ABB RobotStudio station: ExternalGuidedMotion.rsstn

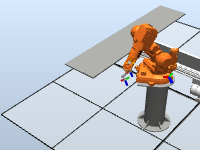
Station E459_norbert (saved by RobotStudio format 3)
Controller IRB140_6kg_0.81m_typeC_1, task T_ROB1: task frame (RAPID world) sits at (10, 680, 720) mm, rotated rx 0 ry 0 rz -30 deg in the station
Controller NorbertEGMVirtuel, task T_ROB1: task frame (RAPID world) sits at (-305, -752, 720) mm, rotated rx 0 ry 0 rz 30 deg in the station
Controller NorbertEGMVirtuel
  mechanical unit ROB_1: Norbert, 6 joints, base frame (0, 0, 0) mm
  mechanical unit CNV1: ?, 1 joints, base frame (0, 0, 0) mm
Controller IRB140_6kg_0.81m_typeC_1
  mechanical unit ROB_1: Rudolf, 6 joints, base frame (0, 0, 0) mm
Layout (positions relative to the parent item):
  - PedestalR [part, from Libraries\Pedestal.rslib] at (10, 680, 0) mm, rotated rx 0 ry 0 rz 150 deg
  - PedestalN [part, from Libraries\Pedestal.rslib] at (-305, -752, 0) mm, rotated rx 0 ry 0 rz -150 deg
  - Windowtable [part]
  - BordR [part, from Libraries\Desk.rslib] at (193.4, 1497.66, 0) mm, rotated rx 0 ry 0 rz -120 deg
  - Norbert [mechanism, from Libraries\IRB140_6_81_C_01.rslib] at (-305, -752, 720) mm, rotated rx 0 ry 0 rz 30 deg; joint values [-2.4777, 0.5946, 0.434, -2.4087, -0.8902, -0.8561] (rad or m)
  - Rudolf [mechanism, from Libraries\IRB140_6_81_C_01.rslib] at (10, 680, 720) mm, rotated rx 0 ry 0 rz -30 deg; joint values [1.249, 0.6446, -0.2193, 0, 1.1455, 1.249] (rad or m)
  - Conveyor [part, from Libraries\Conveyor.rslib] at (-998.97, -64.27, 615.81) mm, rotated rx 90 ry 0 rz -90 deg
  - tSuctionCup [mechanism, from Libraries\tSuctionCup.rslib] at (-444.43, -1188.19, 990.31) mm, rotated rx -146.84 ry 1 rz -95.37 deg
  - Conveyor_2 [part, from Libraries\Conveyor_1.rslib] at (-998.97, -64.27, 615.81) mm, rotated rx 90 ry 0 rz -90 deg
Attachment: BordR is attached to PedestalR
Attachment: tSuctionCup is attached to Norbert / Link6
Station signals: DI doClose, DI doOpen
Station logic (signal -> signal, property => property):
  NorbertEGMVirtuel.doOpen -> ?.diOpen
  NorbertEGMVirtuel.doClose -> ?.diClose
  ?.doClosed -> NorbertEGMVirtuel.diClosed
Targets, tools, work objects and paths stored in the station, written as RAPID:
! task T_ROB1
MODULE EGM_test_analog
  VAR signalao ao_MoveX;
  VAR signalao ao_MoveY;
  VAR signalao ao_MoveZ;
  TASK PERS loaddata load1:=[5,[0,1,0],[1,0,0,0],0,0,0];
  VAR signalao ao_RotX;
  VAR signalao ao_RotY;
  VAR signalao ao_RotZ;
ENDMODULE

! task T_ROB1
MODULE ExternalGuidedMotion
  TASK PERS tooldata tSuctionCup:=[TRUE,[[120,0,57],[0.707106624,-0.000000155,-0.000000251,0.707106939]],[1,[0,0,1],[1,0,0,0],0,0,0]];
  TASK PERS wobjdata TopOfRamp:=[FALSE,TRUE,"",[[0,0,0],[1,0,0,0]],[[83.664,-716.879,531.772],[0.25,0.25,0.933013,-0.0669873]]];
  VAR robtarget startPoint:=[[83.663994925,-716.879172118,531.771925931],[0.369643972,0.239117982,0.892398933,-0.099045793],[-1,-2,0,1],[9E9,9E9,9E9,9E9,9E9,9E9]];
  PROC main()
    MoveJ startPoint,v500,fine,tSuctionCup;
    SetUpEGM;
  ENDPROC
  PROC runEGM()
  ENDPROC
  PROC SetUpEGM()
    runEGM;
  ENDPROC
ENDMODULE

! task T_ROB1
MODULE LINKEDM
  PROC Linked_m()
  ENDPROC
ENDMODULE

